{attribute 'OPC.UA.DA.StructuredType' := '1'}
FUNCTION_BLOCK FB_Machine_LFT EXTENDS FB_BaseMachine IMPLEMENTS I_Machine



VAR_IN_OUT PERSISTENT
	
	stInputs: ST_INPUTS_LFT;
		
	{attribute 'OPC.UA.DA' := '1'}
  	{attribute 'OPC.UA.DA.StructuredType' := '1'}
	fbHandshakeUpstream: 	FB_HandShake_TrayMovement();
		
	{attribute 'OPC.UA.DA' := '1'}
  	{attribute 'OPC.UA.DA.StructuredType' := '1'}
	fbHandshakeDownstream: 	FB_HandShake_TrayMovement();
	
END_VAR



VAR
	
	stTrayCurrent: ST_Tray;
	
	bIsFirstRun: BOOL := TRUE;
	bEnableIgnitionControl: BOOL := TRUE;
	bFirstInputScan: BOOL := TRUE;
	
	
	{attribute 'OPC.UA.DA' := '1'}
  	{attribute 'OPC.UA.DA.StructuredType' := '1'}
	fbServo_Lift: FB_Lift;
	 					
	

		
	{attribute 'OPC.UA.DA' := '1'}
  	{attribute 'OPC.UA.DA.StructuredType' := '1'}														
	fbServo_LiftArm: FB_LiftArm;
		
	
		
	{attribute 'OPC.UA.DA' := '1'}
  	{attribute 'OPC.UA.DA.StructuredType' := '1'}
	fbSensor_PressSwitch:				FB_AutoSwitch();
		
	{attribute 'OPC.UA.DA' := '1'}
  	{attribute 'OPC.UA.DA.StructuredType' := '1'}
	fbSensor_Lift_Home:					FB_AutoSwitch();
		
	{attribute 'OPC.UA.DA' := '1'}
  	{attribute 'OPC.UA.DA.StructuredType' := '1'}
	fbSensor_Lift_Top:					FB_AutoSwitch();
		
	{attribute 'OPC.UA.DA' := '1'}
  	{attribute 'OPC.UA.DA.StructuredType' := '1'}
	fbSensor_Lift_Bottom:				FB_AutoSwitch();
	
		
	{attribute 'OPC.UA.DA' := '1'}
  	{attribute 'OPC.UA.DA.StructuredType' := '1'}
	fbSensor_LiftArm_Home:				FB_AutoSwitch();
		
	{attribute 'OPC.UA.DA' := '1'}
  	{attribute 'OPC.UA.DA.StructuredType' := '1'}
	fbSensor_LiftArm_Extended:			FB_AutoSwitch();
		
	{attribute 'OPC.UA.DA' := '1'}
  	{attribute 'OPC.UA.DA.StructuredType' := '1'}
	fbSensor_LiftArmVacuum:				FB_AutoSwitch();
		
	{attribute 'OPC.UA.DA' := '1'}
  	{attribute 'OPC.UA.DA.StructuredType' := '1'}
	fbSensor_LiftBrake_Left:			FB_AutoSwitch();
		
	{attribute 'OPC.UA.DA' := '1'}
  	{attribute 'OPC.UA.DA.StructuredType' := '1'}
	fbSensor_LiftBrake_Right:			FB_AutoSwitch();
		
	{attribute 'OPC.UA.DA' := '1'}
  	{attribute 'OPC.UA.DA.StructuredType' := '1'}
	fbAutoGreaser:						FB_AutoGreaser();
		
	{attribute 'OPC.UA.DA' := '1'}
  	{attribute 'OPC.UA.DA.StructuredType' := '1'}
	fbValve_Brake:						FB_Valve_ONOFF_woMonitoring(ValveID:= 'BKV', ValveDescr:= 'Brake Solenoid Valve' , Normal_State_NC_1_NO_0:= TRUE);
		
	{attribute 'OPC.UA.DA' := '1'}
  	{attribute 'OPC.UA.DA.StructuredType' := '1'}
	fbValve_Vacuum:						FB_Valve_ONOFF_woMonitoring(ValveID:= 'VPV', ValveDescr:= 'Vacuum Solenoid Valve' , Normal_State_NC_1_NO_0:= TRUE);
		
	
	
	(**
	**		TESTING / SIMULATION VARIABLES
	**)
	
	tgStartSeq: R_TRIG;
	bExt_Step2: BOOL := FALSE;
	bExt_Step8: BOOL := FALSE;
	bPWR_CTRL AT %Q* : BOOL;
	bLOCK_CTRL AT %Q* : BOOL;
	
END_VAR

VAR PERSISTENT
													
	// Package all components into structure & array 
	// ST used for readability
	// Arrray used for iterability 
	stAllComponents: ST_LFTComponents;
	
		
	{attribute 'OPC.UA.DA' := '1'}
  	{attribute 'OPC.UA.DA.StructuredType' := '1'}
	fbInterlocks: 			FB_InterlockManager;
	
	bInProgress: BOOL := FALSE;	//used as a flag to signify that we are in an operation
	
	// Sequences
	//fbSeq_MOVE: 	FB_SequenceMOVE;

	//aSeqs: ARRAY[1..10] OF FB_SequenceBase;	
	
	// Maglock
	
	
END_VAR

IF bIsFirstRun THEN
	devices_init();
	devices_update();
	//sequence_init();
	bIsFirstRun := FALSE;
END_IF


devices_update();
(*
// Scan inputs from OPC
IF stInputs.bParamsInitialised AND bEnableIgnitionControl THEN
	IF bFirstInputScan THEN
		stInputs.stSequenceManager.Sequence_Selected := 1;
		stInputs.stSequenceManager.Sequence_Command := E_SequenceState.STOP;
		fbSequenceManager.selectSequence(Sequence := 1); // main sequence
		fbSequenceManager.stopSequence();
		bFirstInputScan := FALSE;
	END_IF
	scanOPCInputs(Inputs := stInputs ); // only scan if SCADA has set the imputs, otherwise keep persistent or initalised variables
END_IF

*)
// Sequence manager
// fbSeq_MOVE.populateSteps();
// aSeqs[1] := fbSeq_MOVE;
// fbSequenceManager(aSequences := aSeqs);

// Interlocks (make sure this is always called second last (so it overrides any target states set by the sequence manager)
IF GVL.bEnableInterlocks THEN
	interlocks();
END_IF

// Update devices
devices_update();
handshakes();
// sequence();


(**
**		TESTING / SIMULATION VARIABLES
**)

(*
tgStartSeq();
IF tgStartSeq.Q THEN
	fbSequenceManager.selectSequence(Sequence := 1);
	fbSequenceManager.startSequence();
END_IF
*)

METHOD devices_init : BOOL
VAR
	VarInfo : __SYSTEM.VAR_INFO;
	setVarID: INT;
END_VAR
// Hold References to devices in a structure and also an array
// A structure is useful where devices are accessed by name (handy with auto-complete and readability)
// The array is useful for when we want to iterate through all of the devices in the machine and apply a global command (i.e. disable all devices)

// Extract the function block instance name and insert it to each function block
// This enables us to share only the function block name over OPC for nested instances (i.e. sequences, interlock manager)
// The contents of each function block is shared over OPC within the Machine as per heirarchy
// When Ignition needs to retrieve details of devices at the interlock manager and sequence, it simply performs a lookup using the VarID as a key



VarInfo := __VARINFO(fbServo_Lift);
fbServo_Lift.setVarID(VarID := VarInfo.Symbol);

VarInfo := __VARINFO(fbServo_LiftArm);
fbServo_LiftArm.setVarID(VarID := VarInfo.Symbol);

VarInfo := __VARINFO(fbSensor_PressSwitch);
fbSensor_PressSwitch.setVarID(VarID := VarInfo.Symbol);

VarInfo := __VARINFO(fbSensor_Lift_Home);
fbSensor_Lift_Home.setVarID(VarID := VarInfo.Symbol);

VarInfo := __VARINFO(fbSensor_Lift_Top);
fbSensor_Lift_Top.setVarID(VarID := VarInfo.Symbol);

VarInfo := __VARINFO(fbSensor_Lift_Bottom);
fbSensor_Lift_Bottom.setVarID(VarID := VarInfo.Symbol);

VarInfo := __VARINFO(fbSensor_LiftArm_Home);
fbSensor_LiftArm_Home.setVarID(VarID := VarInfo.Symbol);

VarInfo := __VARINFO(fbSensor_LiftArm_Extended);
fbSensor_LiftArm_Extended.setVarID(VarID := VarInfo.Symbol);

VarInfo := __VARINFO(fbSensor_LiftArmVacuum);
fbSensor_LiftArmVacuum.setVarID(VarID := VarInfo.Symbol);

VarInfo := __VARINFO(fbSensor_LiftBrake_Left);
fbSensor_LiftBrake_Left.setVarID(VarID := VarInfo.Symbol);

VarInfo := __VARINFO(fbSensor_LiftBrake_Right);
fbSensor_LiftBrake_Right.setVarID(VarID := VarInfo.Symbol);

VarInfo := __VARINFO(fbAutoGreaser);
fbAutoGreaser.setVarID(VarID := VarInfo.Symbol);

VarInfo := __VARINFO(fbValve_Brake);
fbValve_Brake.setVarID(VarID := VarInfo.Symbol);

VarInfo := __VARINFO(fbValve_Vacuum);
fbValve_Vacuum.setVarID(VarID := VarInfo.Symbol);

aAllComponents[1]  :=  ADR(fbServo_LifT);
aAllComponents[2]  :=  ADR(fbServo_LiftArm);
aAllComponents[3]  :=  ADR(fbSensor_PressSwitch);
aAllComponents[4]  :=  ADR(fbSensor_Lift_Home );
aAllComponents[5]  :=  ADR(fbSensor_Lift_Top );
aAllComponents[6]  :=  ADR(fbSensor_LiftArm_Home  );
aAllComponents[7]  :=  ADR(fbSensor_LiftArm_Extended );
aAllComponents[8]  :=  ADR(fbSensor_LiftArmVacuum );
aAllComponents[9]  :=  ADR(fbSensor_LiftBrake_Left );
aAllComponents[10]  :=  ADR(fbSensor_LiftBrake_Right);
aAllComponents[11]  :=  ADR(fbAutoGreaser);
aAllComponents[12]  :=  ADR(fbValve_Brake);
aAllComponents[13]  :=  ADR(fbValve_Vacuum);
aAllComponents[14]  :=  ADR(fbHandshakeDownstream);
aAllComponents[15]  :=  ADR(fbHandshakeUpstream);



fbServo_LifT.setID(ID := 'Sample ID');									
fbServo_LiftArm.setID(ID := 'Sample ID');
fbSensor_PressSwitch.setID(ID := 'Sample ID');
fbSensor_Lift_Home.setID(ID := 'Sample ID');			
fbSensor_Lift_Top.setID(ID := 'Sample ID');
fbSensor_Lift_Bottom.setID(ID := 'Sample ID');
fbSensor_LiftArm_Home.setID(ID := 'Sample ID');
fbSensor_LiftArm_Extended.setID(ID := 'Sample ID');
fbSensor_LiftArmVacuum.setID(ID := 'Sample ID');
fbSensor_LiftBrake_Left.setID(ID := 'Sample ID');
fbSensor_LiftBrake_Right.setID(ID := 'Sample ID');
fbAutoGreaser.setID(ID := 'Sample ID');			
fbValve_Brake.setID(ID := 'Sample ID');		
fbValve_Vacuum.setID(ID := 'Sample ID');	
fbHandshakeDownstream.setID(ID := 'Downstream tray exchange handshake');
fbHandshakeUpstream.setID(ID := 'Upstream tray exchange handshake');



stAllComponents.fbServo_Lift 				:= ADR(fbServo_Lift);
stAllComponents.fbServo_LiftArm				:= ADR(fbServo_LiftArm);
stAllComponents.fbSensor_PressSwitch		:= ADR(fbSensor_PressSwitch);
stAllComponents.fbSensor_Lift_Home			:= ADR(fbSensor_Lift_Home);
stAllComponents.fbSensor_Lift_Top			:= ADR(fbSensor_Lift_Top);
stAllComponents.fbSensor_Lift_Bottom		:= ADR(fbSensor_Lift_Bottom);
stAllComponents.fbSensor_LiftArm_Home		:= ADR(fbSensor_LiftArm_Home);
stAllComponents.fbSensor_LiftArm_Extended	:= ADR(fbSensor_LiftArm_Extended);
stAllComponents.fbSensor_LiftArmVacuum		:= ADR(fbSensor_LiftArmVacuum);
stAllComponents.fbSensor_LiftBrake_Left		:= ADR(fbSensor_LiftBrake_Left);
stAllComponents.fbSensor_LiftBrake_Right	:= ADR(fbSensor_LiftBrake_Right);
stAllComponents.fbAutoGreaser				:= ADR(fbAutoGreaser);
stAllComponents.fbValve_Brake				:= ADR(fbValve_Brake);
stAllComponents.fbValve_Vacuum				:= ADR(fbValve_Vacuum);


// Note that the soil sensors have not been added to the stAllComponents or components array at this stage
// They are not being used in sequences or interlocks (at this stage)

nQtyComponents := 15;

devices_disable_All();
END_METHOD

METHOD devices_update : BOOL
VAR_INPUT
END_VAR
fbServo_LifT();									
fbServo_LiftArm();
fbSensor_PressSwitch();
fbSensor_Lift_Home();			
fbSensor_Lift_Top();
fbSensor_Lift_Bottom();
fbSensor_LiftArm_Home();
fbSensor_LiftArm_Extended();
fbSensor_LiftArmVacuum();
fbSensor_LiftBrake_Left();
fbSensor_LiftBrake_Right();
fbAutoGreaser();			
fbValve_Brake();		
fbValve_Vacuum();	
fbHandshakeDownstream();
fbHandshakeUpstream();
END_METHOD

METHOD FB_init : BOOL
VAR_INPUT
	bInitRetains : BOOL; // if TRUE, the retain variables are initialized (warm start / cold start)
	bInCopyCode : BOOL;  // if TRUE, the instance afterwards gets moved into the copy code (online change)
	
	ID: STRING;
	Description: STRING;

	
END_VAR
sID := ID;
sDescr := Description;
END_METHOD

METHOD handshakes : BOOL
VAR_INPUT
END_VAR
(*
*
*				DOWNSTREAM HANDSHAKE (we are sending a tray downstream)
*)

(*

IF fbHandshakeDownstream.stTrayExchgangeOutput.eState = E_TrayExchangeState.IDLE AND (fbSensor_TrayEnd.getState() = E_DeviceState.ON) THEN
	fbHandshakeDownstream.stTrayExchangeInput.eState := E_TrayExchangeState.REQUESTED;
END_IF

IF fbHandshakeDownstream.stTrayExchgangeOutput.eState = E_TrayExchangeState.ACCEPTED THEN //AND bTrayisReady THEN
	fbHandshakeDownstream.stTrayExchangeInput.eState := E_TrayExchangeState.IN_PROGRESS;
END_IF

IF fbHandshakeDownstream.stTrayExchgangeOutput.eState = E_TrayExchangeState.COMPLETED THEN
	fbHandshakeDownstream.stTrayExchangeInput.stTrayOutgoing := stTrayCurrent;
END_IF



(*
*
*				UPSTREAM HANDSHAKE (we are receiving a tray)
*)


IF fbHandshakeUpstream.stTrayExchgangeOutput.eState = E_TrayExchangeState.REQUESTED  THEN // bTrayisReady THEN
	fbHandshakeUpstream.stTrayExchangeInput.eState := E_TrayExchangeState.ACCEPTED;
END_IF


IF fbHandshakeUpstream.stTrayExchgangeOutput.eState = E_TrayExchangeState.ACCEPTED THEN // AND bStartingtoMove THEN
	fbHandshakeUpstream.stTrayExchangeInput.eState := E_TrayExchangeState.IN_PROGRESS;
END_IF


IF fbHandshakeUpstream.stTrayExchgangeOutput.eState = E_TrayExchangeState.COMPLETED THEN
	stTrayCurrent := fbHandshakeUpstream.stTrayExchangeInput.stTrayOutgoing;
END_IF

*)
END_METHOD

METHOD interlocks : BOOL
VAR_INPUT
END_VAR
fbInterlocks.init();

(*
fbInterlocks.update(
							Description:= 'Linear Actuator 1 Attempted to Move While Static Conveyor Running',
							InterlockType:= E_InterlockType.RunInterlock, 
							Subject_Device:= ADR(fbLinAct_POP1), 
							Subject_State:= E_DeviceState.IDLE, 
							Signal:=  (fbStaticConv_POP1.getState() = E_DeviceState.RUNNING) OR (fbStaticConv_POP2.getState() = E_DeviceState.RUNNING)
										OR (fbStaticConv_POP3.getState() = E_DeviceState.RUNNING) OR (fbStaticConv_POP1.getState() = E_DeviceState.REVERSE) OR (fbStaticConv_POP2.getState() = E_DeviceState.REVERSE)
										OR (fbStaticConv_POP3.getState() = E_DeviceState.REVERSE),
							HoldSequence:=	FALSE);
							

fbInterlocks.update(
							Description:= 'Linear Actuator 2 Attempted to Move While Static Conveyor Running',
							InterlockType:= E_InterlockType.RunInterlock, 
							Subject_Device:= ADR(fbLinAct_POP2), 
							Subject_State:= E_DeviceState.IDLE, 
							Signal:=  (fbStaticConv_POP1.getState() = E_DeviceState.RUNNING) OR (fbStaticConv_POP2.getState() = E_DeviceState.RUNNING)
										OR (fbStaticConv_POP3.getState() = E_DeviceState.RUNNING) OR (fbStaticConv_POP1.getState() = E_DeviceState.REVERSE) OR (fbStaticConv_POP2.getState() = E_DeviceState.REVERSE)
										OR (fbStaticConv_POP3.getState() = E_DeviceState.REVERSE),
							HoldSequence:=	FALSE);

fbInterlocks.update(
							Description:= 'Linear Actuator 3 Attempted to Move While Static Conveyor Running',
							InterlockType:= E_InterlockType.RunInterlock, 
							Subject_Device:= ADR(fbLinAct_POP3), 
							Subject_State:= E_DeviceState.IDLE, 
							Signal:=  (fbStaticConv_POP1.getState() = E_DeviceState.RUNNING) OR (fbStaticConv_POP2.getState() = E_DeviceState.RUNNING)
										OR (fbStaticConv_POP3.getState() = E_DeviceState.RUNNING) OR (fbStaticConv_POP1.getState() = E_DeviceState.REVERSE) OR (fbStaticConv_POP2.getState() = E_DeviceState.REVERSE)
										OR (fbStaticConv_POP3.getState() = E_DeviceState.REVERSE),
							HoldSequence:=	FALSE);
							
							
fbInterlocks.update(
							Description:= 'Static Conveyor 1 Attemped to Move While POPs Are Moving',
							InterlockType:= E_InterlockType.RunInterlock, 
							Subject_Device:= ADR(fbStaticConv_POP1), 
							Subject_State:= E_DeviceState.IDLE, 
							Signal:=  (fbLinAct_POP1.getState() = E_DeviceState.RUNNING) OR (fbLinAct_POP2.getState() = E_DeviceState.RUNNING)
										OR (fbLinAct_POP3.getState() = E_DeviceState.RUNNING) OR (fbLinAct_POP1.getState() = E_DeviceState.REVERSE) OR (fbLinAct_POP2.getState() = E_DeviceState.REVERSE)
										OR (fbLinAct_POP3.getState() = E_DeviceState.REVERSE),
							HoldSequence:=	FALSE);
							

fbInterlocks.update(
							Description:= 'Static Conveyor 2 Attemped to Move While POPs Are Moving',
							InterlockType:= E_InterlockType.RunInterlock, 
							Subject_Device:= ADR(fbStaticConv_POP2), 
							Subject_State:= E_DeviceState.IDLE, 
							Signal:=  (fbLinAct_POP1.getState() = E_DeviceState.RUNNING) OR (fbLinAct_POP2.getState() = E_DeviceState.RUNNING)
										OR (fbLinAct_POP3.getState() = E_DeviceState.RUNNING) OR (fbLinAct_POP1.getState() = E_DeviceState.REVERSE) OR (fbLinAct_POP2.getState() = E_DeviceState.REVERSE)
										OR (fbLinAct_POP3.getState() = E_DeviceState.REVERSE),
							HoldSequence:=	FALSE);
							

fbInterlocks.update(
							Description:= 'Static Conveyor 3 Attemped to Move While POPs Are Moving',
							InterlockType:= E_InterlockType.RunInterlock, 
							Subject_Device:= ADR(fbStaticConv_POP3), 
							Subject_State:= E_DeviceState.IDLE, 
							Signal:=  (fbLinAct_POP1.getState() = E_DeviceState.RUNNING) OR (fbLinAct_POP2.getState() = E_DeviceState.RUNNING)
										OR (fbLinAct_POP3.getState() = E_DeviceState.RUNNING) OR (fbLinAct_POP1.getState() = E_DeviceState.REVERSE) OR (fbLinAct_POP2.getState() = E_DeviceState.REVERSE)
										OR (fbLinAct_POP3.getState() = E_DeviceState.REVERSE),
							HoldSequence:=	FALSE);	

							
fbInterlocks.update(
							Description:= 'Static Conveyor 1 Attemped to Move When Tray Centre Actuators are Centred',
							InterlockType:= E_InterlockType.RunInterlock, 
							Subject_Device:= ADR(fbStaticConv_POP1), 
							Subject_State:= E_DeviceState.IDLE, 
							Signal:=  (fbTrayCentre_POP1.getState() = E_DeviceState.EXTENDED) OR (fbTrayCentre_POP2.getState() = E_DeviceState.EXTENDED)
										OR (fbTrayCentre_POP3.getState() = E_DeviceState.EXTENDED),
							HoldSequence:=	FALSE);							
							
fbInterlocks.update(
							Description:= 'Static Conveyor 2 Attemped to Move When Tray Centre Actuators are Centred',
							InterlockType:= E_InterlockType.RunInterlock, 
							Subject_Device:= ADR(fbStaticConv_POP2), 
							Subject_State:= E_DeviceState.IDLE, 
							Signal:=  (fbTrayCentre_POP1.getState() = E_DeviceState.EXTENDED) OR (fbTrayCentre_POP2.getState() = E_DeviceState.EXTENDED)
										OR (fbTrayCentre_POP3.getState() = E_DeviceState.EXTENDED),
							HoldSequence:=	FALSE);		
							
							
fbInterlocks.update(
							Description:= 'Static Conveyor 3 Attemped to Move When Tray Centre Actuators are Centred',
							InterlockType:= E_InterlockType.RunInterlock, 
							Subject_Device:= ADR(fbStaticConv_POP3), 
							Subject_State:= E_DeviceState.IDLE, 
							Signal:=  (fbTrayCentre_POP1.getState() = E_DeviceState.EXTENDED) OR (fbTrayCentre_POP2.getState() = E_DeviceState.EXTENDED)
										OR (fbTrayCentre_POP3.getState() = E_DeviceState.EXTENDED),
							HoldSequence:=	FALSE);		
							
							
							
(* HANDSHAKING INTERLOCKS *)
							
fbInterlocks.update(
							Description:= 'Wait for tray RESQUESTED signal',
							InterlockType:= E_InterlockType.RunInterlock, 
							Subject_Device:= ADR(fbStaticConv_POP1), 
							Subject_State:= E_DeviceState.IDLE, 
							Signal:=  ((fbSequenceManager.getCurrentSeq_ID() = E_SequenceList_POP.SEQ_EXTEND_CONVEY) OR
										(fbSequenceManager.getCurrentSeq_ID() = E_SequenceList_POP.SEQ_RETRACT_CONVEY)) AND
										fbHandshakeDownstream.stTrayExchgangeOutput.eState <> E_TrayExchangeState.IN_PROGRESS,
							HoldSequence:=	FALSE);		
							
							
fbInterlocks.update(
							Description:= 'Wait for tray RESQUESTED signal',
							InterlockType:= E_InterlockType.RunInterlock, 
							Subject_Device:= ADR(fbStaticConv_POP2), 
							Subject_State:= E_DeviceState.IDLE, 
							Signal:=  ((fbSequenceManager.getCurrentSeq_ID() = E_SequenceList_POP.SEQ_EXTEND_CONVEY) OR
										(fbSequenceManager.getCurrentSeq_ID() = E_SequenceList_POP.SEQ_RETRACT_CONVEY)) AND
										fbHandshakeDownstream.stTrayExchgangeOutput.eState <> E_TrayExchangeState.IN_PROGRESS,
							HoldSequence:=	FALSE);		

fbInterlocks.update(
							Description:= 'Wait for tray RESQUESTED signal',
							InterlockType:= E_InterlockType.RunInterlock, 
							Subject_Device:= ADR(fbStaticConv_POP3), 
							Subject_State:= E_DeviceState.IDLE, 
							Signal:=  ((fbSequenceManager.getCurrentSeq_ID() = E_SequenceList_POP.SEQ_EXTEND_CONVEY) OR
										(fbSequenceManager.getCurrentSeq_ID() = E_SequenceList_POP.SEQ_RETRACT_CONVEY)) AND
										fbHandshakeDownstream.stTrayExchgangeOutput.eState <> E_TrayExchangeState.IN_PROGRESS,
							HoldSequence:=	FALSE);									
							
fbInterlocks.update(
							Description:= 'Wait for tray RESQUESTED signal',
							InterlockType:= E_InterlockType.RunInterlock, 
							Subject_Device:= ADR(fbLinAct_POP1), 
							Subject_State:= E_DeviceState.IDLE, 
							Signal:=  ((fbSequenceManager.getCurrentSeq_ID() = E_SequenceList_POP.SEQ_CONVEY_EXTEND) OR
										(fbSequenceManager.getCurrentSeq_ID() = E_SequenceList_POP.SEQ_CONVEY_RETRACT)) AND
										fbHandshakeDownstream.stTrayExchgangeOutput.eState <> E_TrayExchangeState.IN_PROGRESS,
							HoldSequence:=	FALSE);		

fbInterlocks.update(
							Description:= 'Wait for tray RESQUESTED signal',
							InterlockType:= E_InterlockType.RunInterlock, 
							Subject_Device:= ADR(fbLinAct_POP2), 
							Subject_State:= E_DeviceState.IDLE, 
							Signal:=  ((fbSequenceManager.getCurrentSeq_ID() = E_SequenceList_POP.SEQ_CONVEY_EXTEND) OR
										(fbSequenceManager.getCurrentSeq_ID() = E_SequenceList_POP.SEQ_CONVEY_RETRACT)) AND
										fbHandshakeDownstream.stTrayExchgangeOutput.eState <> E_TrayExchangeState.IN_PROGRESS,
							HoldSequence:=	FALSE);									

fbInterlocks.update(
							Description:= 'Wait for tray RESQUESTED signal',
							InterlockType:= E_InterlockType.RunInterlock, 
							Subject_Device:= ADR(fbLinAct_POP3), 
							Subject_State:= E_DeviceState.IDLE, 
							Signal:=  ((fbSequenceManager.getCurrentSeq_ID() = E_SequenceList_POP.SEQ_CONVEY_EXTEND) OR
										(fbSequenceManager.getCurrentSeq_ID() = E_SequenceList_POP.SEQ_CONVEY_RETRACT)) AND
										fbHandshakeDownstream.stTrayExchgangeOutput.eState <> E_TrayExchangeState.IN_PROGRESS,
							HoldSequence:=	FALSE);		

*)
fbInterlocks.execute();
END_METHOD

METHOD scanOPCInputs : BOOL
VAR_INPUT
	Inputs: ST_INPUTS_LFT;
END_VAR

VAR 
	nCurrenSeq_Temp: INT;
	nPrev_Seq: INT;
END_VAR

(*
			SEQUENCE CONTROL
*)



IF stInputs.stSequenceManager.Sequence_Selected <> fbSequenceManager.getCurrentSeq_ID() THEN // Selected sequence has been changed
	fbSequenceManager.stopSequence();
	devices_disable_All();
	fbSequenceManager.selectSequence(stInputs.stSequenceManager.Sequence_Selected);
	devices_enable_CurrSeq();
END_IF


IF stInputs.stSequenceManager.Sequence_Ack_Interlock THEN
	fbSequenceManager.acknowledgePause();
	stInputs.stSequenceManager.Sequence_Ack_Interlock := FALSE;
END_IF


CASE stInputs.stSequenceManager.Sequence_Command OF
	E_SequenceState.RUN:
		IF fbSequenceManager.getState() <> E_SequenceState.RUN THEN
			fbSequenceManager.startSequence();
			stInputs.stSequenceManager.Sequence_Command := E_SequenceState.WAIT;
		END_IF
	E_SequenceState.STOP:
		IF fbSequenceManager.getState() <> E_SequenceState.STOP THEN
			fbSequenceManager.stopSequence();
			stInputs.stSequenceManager.Sequence_Command := E_SequenceState.WAIT;
		END_IF
	E_SequenceState.HOLD:
		IF fbSequenceManager.getState() <> E_SequenceState.HOLD THEN
			fbSequenceManager.pauseSequence();
			stInputs.stSequenceManager.Sequence_Command := E_SequenceState.WAIT;
		END_IF
END_CASE

(*
(*
			POP ACTUATORS
*)

fbLinAct_POP1.setMode(Mode := stInputs.stLinAct_POP1.Mode);
IF fbLinAct_POP1.inManual() THEN
	fbLinAct_POP1.setCommand(StateTarget := stInputs.stLinAct_POP1.Command);
ELSE
	stInputs.stLinAct_POP1.Command := fbLinAct_POP1.getCommand();
END_IF


fbLinAct_POP2.setMode(Mode := stInputs.stLinAct_POP2.Mode);
IF fbLinAct_POP2.inManual() THEN
	fbLinAct_POP2.setCommand(StateTarget := stInputs.stLinAct_POP2.Command);
ELSE
	stInputs.stLinAct_POP2.Command := fbLinAct_POP2.getCommand();
END_IF

fbLinAct_POP3.setMode(Mode := stInputs.stLinAct_POP3.Mode);
IF fbLinAct_POP3.inManual() THEN
	fbLinAct_POP3.setCommand(StateTarget := stInputs.stLinAct_POP3.Command);
ELSE
	stInputs.stLinAct_POP3.Command := fbLinAct_POP3.getCommand();
END_IF


(*
			TRAY CENTRE ACTUATORS
*)

fbTrayCentre_POP1.setMode(Mode := stInputs.stTrayCentre_POP1.Mode);
IF fbTrayCentre_POP1.inManual() THEN
	fbTrayCentre_POP1.setCommand(StateTarget := stInputs.stTrayCentre_POP1.Command);
ELSE
	stInputs.stTrayCentre_POP1.Command := fbTrayCentre_POP1.getCommand();
END_IF

fbTrayCentre_POP2.setMode(Mode := stInputs.stTrayCentre_POP2.Mode);
IF fbTrayCentre_POP2.inManual() THEN
	fbTrayCentre_POP2.setCommand(StateTarget := stInputs.stTrayCentre_POP2.Command);
ELSE
	stInputs.stTrayCentre_POP2.Command := fbTrayCentre_POP2.getCommand();
END_IF

fbTrayCentre_POP3.setMode(Mode := stInputs.stTrayCentre_POP3.Mode);
IF fbTrayCentre_POP3.inManual() THEN
	fbTrayCentre_POP3.setCommand(StateTarget := stInputs.stTrayCentre_POP3.Command);
ELSE
	stInputs.stTrayCentre_POP3.Command := fbTrayCentre_POP3.getCommand();
END_IF



(*
			STATIC CONVEYORS
*)


fbStaticConv_POP1.setMode(Mode := stInputs.stStaticConv_POP1.Mode);
IF fbStaticConv_POP1.inManual() THEN
	fbStaticConv_POP1.setCommand(StateTarget := stInputs.stStaticConv_POP1.Command);
ELSE
	stInputs.stStaticConv_POP1.Command := fbStaticConv_POP1.getCommand();
END_IF
									
fbStaticConv_POP2.setMode(Mode := stInputs.stStaticConv_POP2.Mode);
IF fbStaticConv_POP2.inManual() THEN
	fbStaticConv_POP2.setCommand(StateTarget := stInputs.stStaticConv_POP2.Command);
ELSE
	stInputs.stStaticConv_POP2.Command := fbStaticConv_POP2.getCommand();
END_IF

fbStaticConv_POP3.setMode(Mode := stInputs.stStaticConv_POP3.Mode);
IF fbStaticConv_POP3.inManual() THEN
	fbStaticConv_POP3.setCommand(StateTarget := stInputs.stStaticConv_POP3.Command);
ELSE
	stInputs.stStaticConv_POP3.Command := fbStaticConv_POP3.getCommand();
END_IF													


*)
END_METHOD

METHOD sequence : BOOL
VAR_INPUT
END_VAR
(*

IF (fbSequenceManager.getState() = E_SequenceState.COMPLETE) AND (fbHandshakeUpstream.stTrayExchgangeOutput.eState = E_TrayExchangeState.REQUESTED) AND NOT bInProgress THEN
	
	CASE ePOP_Type OF 
		E_POP_Type.EXTEND_CONVEY:
			fbSequenceManager.selectSequence(Sequence := E_SequenceList_POP.SEQ_EXTEND_CONVEY);
		E_POP_Type.CONVEY_EXTEND:
			fbSequenceManager.selectSequence(Sequence := E_SequenceList_POP.SEQ_CONVEY_EXTEND);
		E_POP_Type.RETRACT_CONVEY:
			fbSequenceManager.selectSequence(Sequence := E_SequenceList_POP.SEQ_RETRACT_CONVEY);
		E_POP_Type.CONVEY_RETRACT:
			fbSequenceManager.selectSequence(Sequence := E_SequenceList_POP.SEQ_RETRACT_CONVEY);
	END_CASE

	fbSequenceManager.startSequence();
	bInProgress := TRUE;
END_IF



IF (fbSequenceManager.getState() = E_SequenceState.COMPLETE) AND bInProgress THEN
	// return the pop conveyor back to resting condition
	CASE ePOP_Type OF 
		E_POP_Type.EXTEND_CONVEY:
			fbSequenceManager.selectSequence(Sequence := E_SequenceList_POP.SEQ_RETRACT);
		E_POP_Type.CONVEY_EXTEND:
			fbSequenceManager.selectSequence(Sequence := E_SequenceList_POP.SEQ_RETRACT);
		E_POP_Type.RETRACT_CONVEY:
			fbSequenceManager.selectSequence(Sequence := E_SequenceList_POP.SEQ_EXTEND);
		E_POP_Type.CONVEY_RETRACT:
			fbSequenceManager.selectSequence(Sequence := E_SequenceList_POP.SEQ_EXTEND);
	END_CASE
	fbSequenceManager.startSequence();
	bInProgress := FALSE;
END_IF

*)
END_METHOD

METHOD sequence_init : BOOL
VAR_INPUT
END_VAR
(*fbSeq_MOVE(devices := stAllComponents, bExt_1_Ret_0_Step2 := bExt_Step2, bExt_1_Ret_0_Step8 := bExt_Step8);
fbSeq_MOVE.populateSteps();
aSeqs[1] := fbSeq_MOVE;
*)
(*
fbSeq_RET_CONV(devices := stAllComponents);
fbSeq_CONV_EXT(devices := stAllComponents);
fbSeq_CONV_RET(devices := stAllComponents);
fbSeq_EXT(devices := stAllComponents);
fbSeq_RET(devices := stAllComponents);
*)


(*
fbSeqRND_DMMain(devices := stAllComponents);
fbSeqRND_DMCal(devices := stAllComponents);
fbSeqRND_DMFill(devices := stAllComponents);
fbSeqRND_DMDrain(devices := stAllComponents);
fbSeqRND_DMFlush(devices := stAllComponents);

fbSeqRND_DMMain.populateSteps();
fbSeqRND_DMCal.populateSteps();
fbSeqRND_DMFill.populateSteps();
fbSeqRND_DMDrain.populateSteps();
fbSeqRND_DMFlush.populateSteps();

aSeqs[1] := fbSeqRND_DMMain;
aSeqs[2] := fbSeqRND_DMCal;
aSeqs[3] := fbSeqRND_DMFill;
aSeqs[4] := fbSeqRND_DMDrain;
aSeqs[5] := fbSeqRND_DMFlush;


*)
END_METHOD

END_FUNCTION_BLOCK

(* stored: Version 1.1.0.1, ProductVersion 3.1.4024.12
   POU FB_Machine_LFT: Id {dd0b1c07-301a-41cb-aaee-ff837cc40ded}, SpecialFunc None
   Method devices_init: Id {a68727a6-fad2-4558-8640-42f72ece9114}
   Method devices_update: Id {1b7feb4b-cbbc-4c6a-b389-6856fb398443}
   Method FB_init: Id {9859e583-9672-4a64-b482-d0b6ecf9ad87}
   Method handshakes: Id {6deb0032-ab07-4713-b463-7cc1bc65b2d6}
   Method interlocks: Id {59193bb1-61de-46c6-9e61-e4b5fd0dffc1}
   Method scanOPCInputs: Id {4ab94a57-734f-492b-b7ca-b018517c8a45}
   Method sequence: Id {682d83a0-ee3a-4a43-a046-60c8c29d9f33}
   Method sequence_init: Id {41dd3da2-5c40-4f9d-8304-c735973b9623} *)
